FUNCTION_BLOCK FB_IotMqttCommunication
VAR_INPUT
	sTopicToPublish: STRING(255); // MQTT topic
    sMessageToPublish: STRING(255); // Message buffer

END_VAR
VAR_OUTPUT
END_VAR
VAR
	fbMqttClient: FB_IotMqttClient;
	bInitSent : BOOL := FALSE;
	tmrSendMessageInterval: TON := (PT := T#10S); // Interval timer for publishing
END_VAR

fbMqttClient.sHostName := '158.180.44.197';
fbMqttClient.nHostPort := 1883;
fbMqttClient.sTopicPrefix := 'aut/DerGeraet/';
fbMqttClient.sClientId := 'Publishing PLC';
fbMqttClient.sUserName := 'bobm';
fbMqttClient.sUserPassword := 'letmein';
     // MQTT client with initialization
	

fbMqttClient.Execute(bConnect := TRUE);

IF fbMqttClient.bConnected THEN
    tmrSendMessageInterval(IN := TRUE);
	
	IF NOT bInitSent THEN //Init messagees 
		//send Group name
        fbMqttClient.Publish(
            sTopic := '$$groupname',
            pPayload := ADR('DerGreraet'),
            nPayloadSize := LEN('DerGreraet') + 1,
            eQoS := TcIotMqttQos.AtMostOnceDelivery,
            bRetain := TRUE,
            bQueue := FALSE
        );	
		//send group members
        fbMqttClient.Publish(
            sTopic := 'names',
            pPayload := ADR('Naidr, Schulte, Brandt'),
            nPayloadSize := LEN('Naidr, Schulte, Brandt') + 1,
            eQoS := TcIotMqttQos.AtMostOnceDelivery,
            bRetain := TRUE,
            bQueue := FALSE
        );	
		//send unit
        fbMqttClient.Publish(
            sTopic := 'bEnable/$$unit',
            pPayload := ADR('BOOL'),
            nPayloadSize := LEN('BOOL') + 1,
            eQoS := TcIotMqttQos.AtMostOnceDelivery,
            bRetain := TRUE,
            bQueue := FALSE
        );
		bInitSent := TRUE;
	END_IF
	
    IF tmrSendMessageInterval.Q THEN
        tmrSendMessageInterval(IN := FALSE);

        fbMqttClient.Publish(
            sTopic := sTopicToPublish,
            pPayload := ADR(sMessageToPublish),
            nPayloadSize := LEN(sMessageToPublish) + 1,
            eQoS := TcIotMqttQos.AtMostOnceDelivery,
            bRetain := FALSE,
            bQueue := FALSE
        );
    END_IF
END_IF

END_FUNCTION_BLOCK

(* stored: Version 1.1.0.1, ProductVersion 3.1.4024.15
   POU FB_IotMqttCommunication: Id {50763065-5558-483e-9e3a-6575a5829d35}, SpecialFunc None *)
